INTERFACE ITF_ControlElement4 EXTENDS ITF_BaseControlElement

END_INTERFACE

(* stored: Version 1.1.0.1, ProductVersion 3.1.4024.15
   Itf ITF_ControlElement4: Id {b9349418-826d-44cb-856f-f8c002f53398} *)
